// TIA Portal V20 export
TYPE "LER_typeRadiusMeasureInterface"
// stored: Access Published
   STRUCT
      commands : "LER_typeRadiusMeasureCommnads";
      monitoring : "LER_typeRadiusMeasureMonitioing";
      configuration : "LER_typeRadiusMeasureConfiguration";
   END_STRUCT;
END_TYPE
